# B&R Automation Studio project Lib_MathTools
Automation Studio 4.7.3.93 SP

## Configuration ARsim

CPU PC_any, AutomationRuntime C4.72, Build 4.1.2, Vc V4.72.0

### Task classes (Cpu.sw)
```
Cyclic#4:
  Example <- Example.prg
Libraries: MathTools
```

### Hardware
```
PC : PC_any v1.1.0.0 (OrderNumber=PC)
```

## Logical view

Binary libraries used (declarations not repeated): operator, runtime, astime, AsIecCon

### Package Logical/Libraries - Global libraries

### Library Logical/Libraries/MathTools (ANSIC, version 0.01.2) - Miscellaneous math functions

#### MathTools.fun - Exported functions and function blocks
```iecst
(*Integer wrap*)

FUNCTION Math_WrapUSINT : USINT
	VAR_INPUT
		Value : DINT;
		LowerBound : DINT;
		UpperBound : DINT;
	END_VAR
END_FUNCTION

FUNCTION Math_WrapSINT : SINT
	VAR_INPUT
		Value : DINT;
		LowerBound : DINT;
		UpperBound : DINT;
	END_VAR
END_FUNCTION

FUNCTION Math_WrapUINT : UINT
	VAR_INPUT
		Value : DINT;
		LowerBound : DINT;
		UpperBound : DINT;
	END_VAR
END_FUNCTION

FUNCTION Math_WrapINT : INT
	VAR_INPUT
		Value : DINT;
		LowerBound : DINT;
		UpperBound : DINT;
	END_VAR
END_FUNCTION
(*Floating point wrap*)

FUNCTION Math_WrapREAL : REAL
	VAR_INPUT
		Value : LREAL;
		LowerBound : LREAL;
		UpperBound : LREAL;
	END_VAR
END_FUNCTION

FUNCTION Math_WrapLREAL : LREAL
	VAR_INPUT
		Value : LREAL;
		LowerBound : LREAL;
		UpperBound : LREAL;
	END_VAR
END_FUNCTION
(*Quadtratic formula*)

FUNCTION Math_2ndOrderRoots : USINT
	VAR_INPUT
		p2 : LREAL;
		p1 : LREAL;
		p0 : LREAL;
	END_VAR
	VAR_IN_OUT
		Solution : Math2ndOrderRootsSoln_typ;
	END_VAR
END_FUNCTION
(*Heaviside function*)

FUNCTION Math_UnitStep : REAL
	VAR_INPUT
		Input : LREAL;
	END_VAR
END_FUNCTION
```

#### math_tools.c
```c
/*********************************************************************************
 * Copyright: B&R Industrial Automation
 * Author:    Tyler Matijevich
 * Created:   May 14, 2020/1:34 PM
 *********************************************************************************/

#include "MathTools.h"
#include <math.h>

/*
 * Internal function
 * Utilize the implicit conversion from chars/shorts to longs
 */
static signed long WrapInteger(signed long inputValue, signed long lowerBound, signed long upperBound) {
	/* Static functions are functions only visible to other functions in the file */

	if(lowerBound <= upperBound) {
		signed long total 		= upperBound - lowerBound + 1;
		signed long distance 	= inputValue - lowerBound;
		signed long offset 		= distance % total;

		if(offset >= 0)
			return lowerBound + offset;
		else
			return upperBound + offset + 1; // +1 to include the upper bound during subtraction
	}

	else
		return 0;

}

/*
 * Each function will return zero if the bounds exceed data type limits
 * or the lower bound exceeds the upper bound
 */

/* USINT wrap */
unsigned char Math_WrapUSINT(signed long Value, signed long LowerBound, signed long UpperBound) {
	if(LowerBound < 0 || LowerBound > 255 || UpperBound < 0 || UpperBound > 255)
		return 0;
	else
		return (unsigned char)WrapInteger(Value, LowerBound, UpperBound);
}

/* SINT wrap */
signed char Math_WrapSINT(signed long Value, signed long LowerBound, signed long UpperBound) {
	if(LowerBound < -128 || LowerBound > 127 || UpperBound < -128 || UpperBound > 127)
		return 0;
	else
		return (signed char)WrapInteger(Value, LowerBound, UpperBound);
}

/* UINT wrap */
unsigned short Math_WrapUINT(signed long Value, signed long LowerBound, signed long UpperBound) {
	if(LowerBound < 0 || LowerBound > 65535 || UpperBound < 0 || UpperBound > 65535)
		return 0;
	else
		return (unsigned short)WrapInteger(Value, LowerBound, UpperBound);
}

/* INT wrap */
signed short Math_WrapINT(signed long Value, signed long LowerBound, signed long UpperBound) {
	if(LowerBound < -32768 || LowerBound > 32767 || UpperBound < -32768 || UpperBound > 32767)
		return 0;
	else
		return (signed short)WrapInteger(Value, LowerBound, UpperBound);
}

/*
 * Internal function
 * Utilize the implicit conversion from floats to doubles
 */
double WrapDouble(double inputValue, double lowerBound, double upperBound) {
	if(upperBound > lowerBound){
		double distance = inputValue - lowerBound;
		double total = upperBound - lowerBound;
		double offset = distance - trunc(distance / total) * total;
		return (distance >= 0.0)? (lowerBound + offset) : (upperBound + offset);
	} else
		return 0.0;
}

/* REAL wrap */
float Math_WrapREAL(double Value, double LowerBound, double UpperBound) {
	return (float)WrapDouble(Value, LowerBound, UpperBound);
}

/* LREAL wrap */
double Math_WrapLREAL(double Value, double LowerBound, double UpperBound) {
	return WrapDouble(Value, LowerBound, UpperBound);
}

/* 2nd Order Roots (Quadratic formula) $$ p2 * x^2 + p1 * x + p0 = 0 $$ */
plcbit Math_2ndOrderRoots(double p2, double p1, double p0, struct Math2ndOrderRootsSoln_typ* Solution) {
	Solution->r1 = Solution->r2 = 0.0; /* Default/Invalid solution */
	double determinant = pow(p1, 2.0) - 4.0 * p2 * p0;

	if(fabs(p2) > 0.0) { /* Two roots - protect against divide by zero */
		if(determinant > 0.0) {
			Solution->r1 = ((-p1) + sqrt(determinant)) / (2.0 * p2);
			Solution->r2 = ((-p1) - sqrt(determinant)) / (2.0 * p2);
		}

		else if(determinant < 0.0)
			return 0; /* Imaginary roots, do not consider this case */

		else {
			Solution->r1 = (-p1) / (2.0 * p2);
			Solution->r2 = Solution->r1;
		}
		return 1;

	} else {
		if(fabs(p1) > 0.0) { /* One root - protect against divide by zero */
			Solution->r1 = (-p0) / p1;
			Solution->r2 = Solution->r1;
			return 1;

		} else /* No solution */
			return 0;
	}
}

/* Heaviside function */
float Math_UnitStep(double Input){
	return (Input >= 0.0)? 1.0 : 0.0;
}
```

#### mathtools.c - not listed in the package file held
```c
#include "MathTools.h"

/* Internal function */
static signed long fnWrapInteger(signed long inputValue, signed long lowerBound, signed long upperBound) {
	/* Static functions are functions only visible to other functions in the file */

	if(lowerBound <= upperBound) {
		signed long total 		= upperBound - lowerBound + 1;
		signed long distance 	= inputValue - lowerBound;
		signed long offset 		= distance % total;

		if(offset >= 0)
			return lowerBound + offset;
		else
			return upperBound + offset + 1; // +1 to include the upper bound during subtraction
	}

	else
		return 0;

}

/*
 * Each function will return zero if the bounds exceed data type limits
 * or the lower bound exceeds the upper bound
 */

/* USINT wrap */
unsigned char fnWrapUSINT(signed long Value, signed long LowerBound, signed long UpperBound) {
	if(LowerBound < 0 || LowerBound > 255 || UpperBound < 0 || UpperBound > 255)
		return 0;
	else
		return (unsigned char)fnWrapInteger(Value, LowerBound, UpperBound);
}

/* SINT wrap */
signed char fnWrapSINT(signed long Value, signed long LowerBound, signed long UpperBound) {
	if(LowerBound < -128 || LowerBound > 127 || UpperBound < -128 || UpperBound > 127)
		return 0;
	else
		return (signed char)fnWrapInteger(Value, LowerBound, UpperBound);
}

/* UINT wrap */
unsigned short fnWrapUINT(signed long Value, signed long LowerBound, signed long UpperBound) {
	if(LowerBound < 0 || LowerBound > 65535 || UpperBound < 0 || UpperBound > 65535)
		return 0;
	else
		return (unsigned short)fnWrapInteger(Value, LowerBound, UpperBound);
}

/* INT wrap */
signed short fnWrapINT(signed long Value, signed long LowerBound, signed long UpperBound) {
	if(LowerBound < -32768 || LowerBound > 32767 || UpperBound < -32768 || UpperBound > 32767)
		return 0;
	else
		return (signed short)fnWrapInteger(Value, LowerBound, UpperBound);
}
```

### Program Logical/Example (IEC)

#### Variables.var
```iecst
(*Wrap value onto range*)
VAR
	In1 : USINT;
	In2 : SINT;
	In3 : UINT;
	In4 : INT;
	In5 : REAL;
	In6 : LREAL;
	Out1 : USINT;
	Out2 : SINT;
	Out3 : UINT;
	Out4 : INT;
	Out5 : REAL;
	Out6 : LREAL;
END_VAR
(*Quadratic formula*)
VAR
	p2 : REAL;
	p1 : REAL;
	p0 : REAL;
	SolnRoots : Math2ndOrderRootsSoln_typ;
	statusRoots : USINT;
END_VAR
(*Unit step (heaviside) function*)
VAR
	In7 : REAL;
	Out7 : REAL;
END_VAR
```

#### Main.st
```iecst
(*******************************************************************************
 * Copyright: B&R Industrial Automation
 * Author:    Tyler Matijevich
 * Created:   May 14, 2020/11:24 AM
********************************************************************************
 * Description: Example program for MathTools user library
********************************************************************************)

PROGRAM _INIT

	In1 := 5;
	In2 := 1;
	In3 := 1200;
	In4 := -1400;
	In5 := 734.0;
	In6 := -12.0;

	p2 := 2.0;
	p1 := -1.0;
	p0 := -6.0;

	In7 := -1.0;

END_PROGRAM

PROGRAM _CYCLIC

	Out1 := Math_WrapUSINT(In1, 1, 4);
	Out2 := Math_WrapSINT(In2, -3, 0);
	Out3 := Math_WrapUINT(In3, 1, 1000);
	Out4 := Math_WrapINT(In4, -1200, -1);
	Out5 := Math_WrapREAL(In5, 0.0, 360.0);
	Out6 := Math_WrapLREAL(In6, 0.0, 1000.0);

	statusRoots := Math_2ndOrderRoots(p2, p1, p0, SolnRoots);

	Out7 := Math_UnitStep(In7);

END_PROGRAM

PROGRAM _EXIT

END_PROGRAM
```

Listed in the project but not available here: Logical/Global.typ, Logical/Global.var, Logical/Libraries/MathTools/Types.typ, Logical/Libraries/MathTools/Constants.var
